{attribute 'pack_mode' := '1'}
TYPE ST_AddTrafficLightDataOut :
STRUCT
	// Fixed data for all methods
	nNumberOfOutputArguments	: UDINT; // determined amount of output parameters
	nReserved					: ARRAY[1..4] OF BYTE; // Reserved padding
	
	// Method specific data
	stOutputArgInfo				: ARRAY[1..2] OF ST_UAMethodArgInfo; // number of output parameters - M_Mul has 1 output parameter 
	eStatus						: E_MMServerStatus;
	sMessage					: STRING;

END_STRUCT
END_TYPE

(* stored: Version 1.1.0.1, ProductVersion 3.1.4024.5
   DUT ST_AddTrafficLightDataOut: Id {a6bc47fe-05b3-42ca-abe4-73179ba4a7a1} *)
